FUNCTION_BLOCK FB_FullCycleTime
VAR_INPUT
	bPalletSensor			:BOOL;
	timTimeMax				:TIME:= T#120S;
END_VAR
VAR_OUTPUT
	nCurrentCycleTime		:REAL;
	arrCycleTimes			:ARRAY [1..10] OF REAL;
END_VAR
VAR
	tCycleTime				:TON;
	rStart					:R_TRIG;
END_VAR

rStart(CLK:= bPalletSensor);
tCycleTime(IN:= TRUE, PT:= timTimeMax);

IF 		rStart.Q THEN
				MEMMOVE(ADR(arrCycleTimes)+4,ADR(arrCycleTimes),SIZEOF(arrCycleTimes)-4);
				arrCycleTimes[1] := nCurrentCycleTime;
				tCycleTime(IN:= FALSE);
ELSIF	NOT tCycleTime.Q THEN
				nCurrentCycleTime := (TIME_TO_REAL(tCycleTime.ET) / 1000);
ELSE
				nCurrentCycleTime := (TIME_TO_REAL(timTimeMax) / 1000);
END_IF

END_FUNCTION_BLOCK

(* stored: Version 1.1.0.1, ProductVersion 3.1.4024.11
   POU FB_FullCycleTime: Id {22fe7cd3-be76-406a-a8f8-6dd4765a53d7}, SpecialFunc None *)
